
FUNCTION CB_byte_to_bool : BOOL


TITLE = ' Convert a byte into a boolean '
VERSION : '1.0'
AUTHOR  : CB
NAME    : byteToBo
FAMILY  : TNI

VAR_INPUT
    IN : BYTE;
END_VAR

BEGIN

CB_byte_to_bool := (IN <>0);

END_FUNCTION
